TYPE sSmartGreiferProzessVariablen :
STRUCT
	Pos				:USINT;			// Position von Greifer in mm
	Geschw			:USINT;			// Geschwindigkeit in %
	F				:USINT;			// Kraft in %
END_STRUCT
	
END_TYPE

(* stored: Version 1.1.0.1
   DUT sSmartGreiferProzessVariablen: Id {49eaff3b-61aa-4147-8aa0-518a9c2da521} *)
